Fanuc KAREL source: userClear.kl

PROGRAM userClear
%NOBUSYLAMP
%NOLOCKGROUP


%from display.klh %import clear

BEGIN
	display__clear
END userClear
